INTERFACE IBuffer

PROPERTY NumOfItems : DINT
GET
END_GET
END_PROPERTY

PROPERTY BufferFull : BOOL
GET
END_GET
END_PROPERTY

PROPERTY MaxCapacity : DINT
GET
END_GET
END_PROPERTY

END_INTERFACE

(* stored: Version 1.1.0.1, ProductVersion 3.1.0.26
   Itf IBuffer: Id {6ca8dc5e-3ccb-42a7-b725-bd82639cabe8}
   Property NumOfItems: Id {20de0e0f-413e-48f7-9eb2-454894ca89b9}
   Get Get: Id {ccd1eed7-2420-4e9c-93aa-12581d89cd25}
   Property BufferFull: Id {2de9695e-388c-467a-9d08-172885753681}
   Get Get: Id {7d3d5435-71d2-40b6-81bc-99f79e8ae48c}
   Property MaxCapacity: Id {3a32b318-0096-428a-9049-f4cfb01a1120}
   Get Get: Id {fbd5796f-1399-44a8-ab39-d4ee66b2f3df} *)
